FUNCTION_BLOCK controller
  (* Standard: 61499-2 *)
  (* Version 0.1, 2017-00-12, hpea485, UOA *)
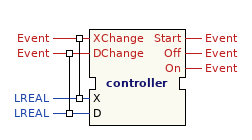
  EVENT_INPUT
    XChange WITH X;
    DChange WITH D;
  END_EVENT
  EVENT_OUTPUT
    Start;
    Off;
    On;
  END_EVENT
  VAR_INPUT
    X : LREAL;
    D : LREAL;
  END_VAR
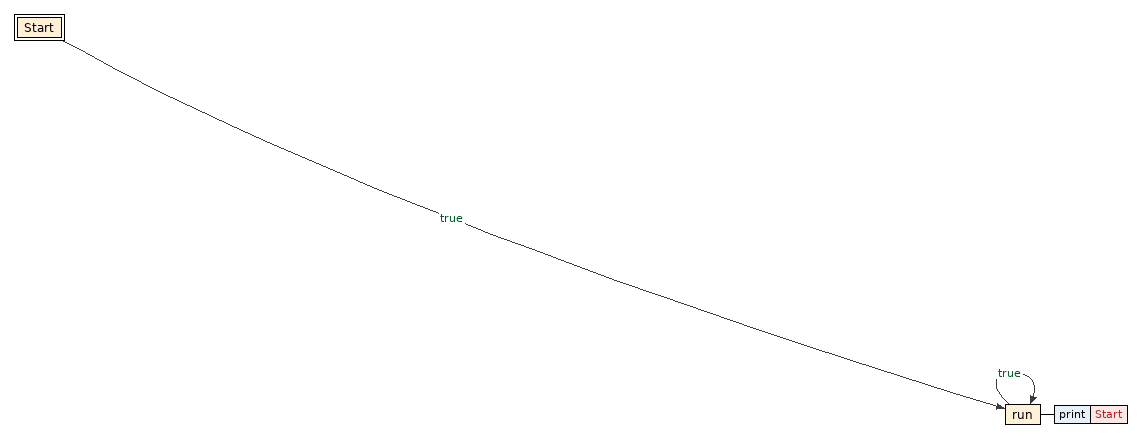
  EC_STATES
    Start;
    run : print -> Start;
  END_STATES
  EC_TRANSITIONS
    Start TO run := true;
    run TO run := true;
  END_TRANSITIONS
  ALGORITHM print IN C:
static int count = 0;

printf("X: %f, D: %f\n", me->X, me->D);

count++;
if(count == 25) {
	me->outputEvents.event.On = 1;
}
if(count == 50) {
	me->outputEvents.event.Off = 1;
	count = 0;
}
  END_ALGORITHM
END_FUNCTION_BLOCK
